{attribute 'TcCallAfterOutputUpdate'}
PROGRAM MAIN
VAR
END_VAR

P_DIOC();

END_PROGRAM

(* stored: Version 1.1.0.1, ProductVersion 3.1.4024.6
   POU MAIN: Id {0b915060-8242-4db1-90e7-448aaf73892f}, SpecialFunc None *)
